{attribute addProperty BoxType "AX8810-0000-0017"}
{attribute addProperty Id "PSM_StatuswordAT %I*PSM_Statusword_B057017B1620WcStateAT %I*WcState_98A4DF7520.250InfoDataAT %I*InfoData_0BDED7BF144180"}
{attribute addProperty CRC "356712783"}
{attribute addProperty SizeInBites "162"}
{attribute addProperty SizeInBytes "20.25"}
TYPE AX8810_B7ACDB90 :
STRUCT
	{attribute addProperty Name "PSM_Statusword"}
	PSM_Statusword : PSM_Statusword_B057017B;
	{attribute addProperty Name "WcState"}
	WcState : WcState_98A4DF75;
	{attribute addProperty Name "InfoData"}
	InfoData : InfoData_0BDED7BF;
END_STRUCT
END_TYPE

(* stored: Version 1.2.0.0, ProductVersion 3.1.4024.9
   DUT AX8810_B7ACDB90: Id {7f0e81ee-64f9-4a3b-938a-62c84a50970d} *)
